TYPE DiDiag :
STRUCT
	{attribute addProperty Name "Diag"}
	Diag AT %I* : BOOL;
END_STRUCT
END_TYPE

(* stored: Version 1.1.0.1, ProductVersion 3.1.4024.9
   DUT DiDiag: Id {360d213f-1d33-046e-0bbc-e479c2b78620} *)
